FUNCTION_BLOCK FB_SignalHandlingIntern IMPLEMENTS I_SignalHandling
VAR_INPUT
	bInput				: BOOL;			// Input signal, e.g. sensor signal, enable for fuse
END_VAR
VAR_OUTPUT
	bOut				: BOOL;			// Processed output signal, e.g. delayed, inverted
END_VAR
VAR
	bEnableLocal		: BOOL;			// Enable processing of input signal
END_VAR

// =========================================================
;
// =========================================================

METHOD Enable
VAR_INPUT
	bEnable		: BOOL;
END_VAR
// =========================================================
// Store input in local variable

	bEnableLocal := bEnable;

// =========================================================
END_METHOD

METHOD SetOutput
VAR_INPUT
END_VAR
// =========================================================

bOut := bInput AND bEnableLocal;

// =========================================================
END_METHOD

END_FUNCTION_BLOCK

(* stored: Version 1.1.0.1, ProductVersion 3.1.4018.2
   POU FB_SignalHandlingIntern: Id {b8b92a6e-c554-43f8-a635-2a73803f1234}, SpecialFunc None
   Method Enable: Id {72c4bf9e-6aed-4efb-85fd-5fe71ec34b14}
   Method SetOutput: Id {fea80c04-4b34-4b2a-8a8e-d9ffa3503a31} *)
